# B&R Automation Studio project RS15_RX_30005_r00 (part 10)

#### HGWeber.fun - Exported functions and function blocks
```iecst
(********************************************************************
 * COPYRIGHT --
 ********************************************************************
 * Library: HGWeber
 * File: HGWeber.fun
 * Author: pkiel
 * Created: September 03, 2009
 ********************************************************************
 * Functions and function blocks of library HGWeber
 ********************************************************************)

FUNCTION H_FC_Modulus_V0 : REAL  (*Calculat the modulus of number*)
  VAR_INPUT
    IN_rMod : REAL ;
    IN_rVar : REAL ;
  END_VAR
  VAR
    rVar : REAL;
  END_VAR
END_FUNCTION

FUNCTION H_FC_Modulus : REAL  (*Calculat the modulus of number*)
  VAR_INPUT
    IN_rMod : REAL ;
    IN_rVar : REAL ;
  END_VAR
  VAR
    rVar : REAL;
  END_VAR
END_FUNCTION

FUNCTION_BLOCK HGW_2StatePB (*Two State Pushbutton Control/Indication*)
	VAR_INPUT
		PB : BOOL; (*Add your parameter comment*)
		Reset : BOOL; (*Add your parameter comment*)
		BackColor_State0 : UINT; (*Add your parameter comment*)
		ForeColor_State0 : UINT; (*Add your parameter comment*)
		BackColor_State1 : UINT; (*Add your parameter comment*)
		ForeColor_State1 : UINT; (*Add your parameter comment*)
	END_VAR
	VAR_OUTPUT
		Text_Ind : UINT; (*Add your parameter comment*)
		Color_Ind : UINT; (*Add your parameter comment*)
		State0 : BOOL; (*Add your parameter comment*)
		State1 : BOOL; (*Add your parameter comment*)
	END_VAR
	VAR
		R_Trig1 : r_trig;
	END_VAR
END_FUNCTION_BLOCK

FUNCTION_BLOCK HGW_3StatePB (*Three State Pushbutton Control/Indication*)
	VAR_INPUT
		PB : BOOL; (*Add your parameter comment*)
		Reset : BOOL; (*Add your parameter comment*)
		BackColor_State0 : UINT; (*Add your parameter comment*)
		ForeColor_State0 : UINT; (*Add your parameter comment*)
		BackColor_State1 : UINT; (*Add your parameter comment*)
		ForeColor_State1 : UINT; (*Add your parameter comment*)
		BackColor_State2 : UINT;
		ForeColor_State2 : UINT;
	END_VAR
	VAR_OUTPUT
		Text_Ind : UINT; (*Add your parameter comment*)
		Color_Ind : UINT; (*Add your parameter comment*)
		State0 : BOOL; (*Add your parameter comment*)
		State1 : BOOL; (*Add your parameter comment*)
		State2 : BOOL; (*Add your parameter comment*)
	END_VAR
	VAR
		R_Trig1 : r_trig;
	END_VAR
END_FUNCTION_BLOCK

FUNCTION_BLOCK HGW_4StatePB (*Four State Pushbutton Control/Indication*)
	VAR_INPUT
		PB : BOOL; (*Add your parameter comment*)
		Reset : BOOL; (*Add your parameter comment*)
		BackColor_State0 : UINT; (*Add your parameter comment*)
		ForeColor_State0 : UINT; (*Add your parameter comment*)
		BackColor_State1 : UINT; (*Add your parameter comment*)
		ForeColor_State1 : UINT; (*Add your parameter comment*)
		BackColor_State2 : UINT; (*Add your parameter comment*)
		ForeColor_State2 : UINT; (*Add your parameter comment*)
		BackColor_State3 : UINT; (*Add your parameter comment*)
		ForeColor_State3 : UINT; (*Add your parameter comment*)
	END_VAR
	VAR_OUTPUT
		Text_Ind : UINT; (*Add your parameter comment*)
		Color_Ind : UINT; (*Add your parameter comment*)
		State0 : BOOL; (*Add your parameter comment*)
		State1 : BOOL; (*Add your parameter comment*)
		State2 : BOOL; (*Add your parameter comment*)
		State3 : BOOL; (*Add your parameter comment*)
	END_VAR
	VAR
		R_Trig1 : r_trig;
	END_VAR
END_FUNCTION_BLOCK

FUNCTION_BLOCK HGW_2StateIND (*Two State Indication*)
	VAR_INPUT
		In_State : BOOL; (*Add your parameter comment*)
		BackColor_State0 : UINT; (*Add your parameter comment*)
		ForeColor_State0 : UINT; (*Add your parameter comment*)
		BackColor_State1 : UINT; (*Add your parameter comment*)
		ForeColor_State1 : UINT; (*Add your parameter comment*)
	END_VAR
	VAR_OUTPUT
		Text_Ind : UINT; (*Add your parameter comment*)
		Color_Ind : UINT; (*Add your parameter comment*)
		State0 : BOOL; (*Add your parameter comment*)
		State1 : BOOL; (*Add your parameter comment*)
	END_VAR
END_FUNCTION_BLOCK

FUNCTION_BLOCK HGW_3StateIND (*Three State Indication*)
  VAR_INPUT
    In_State0 : BOOL; (*Add your parameter comment*)
    In_State1 : BOOL; (*Add your parameter comment*)
    In_State2 : BOOL; (*Add your parameter comment*)
    BackColor_State0 : UINT; (*Add your parameter comment*)
    ForeColor_State0 : UINT; (*Add your parameter comment*)
    BackColor_State1 : UINT; (*Add your parameter comment*)
    ForeColor_State1 : UINT; (*Add your parameter comment*)
    BackColor_State2 : UINT; (*Add your parameter comment*)
    ForeColor_State2 : UINT; (*Add your parameter comment*)
  END_VAR
  VAR_OUTPUT
    Text_Ind : UINT; (*Add your parameter comment*)
    Color_Ind : UINT; (*Add your parameter comment*)
    State0 : BOOL; (*Add your parameter comment*)
    State1 : BOOL; (*Add your parameter comment*)
    State2 : BOOL; (*Add your parameter comment*)
  END_VAR
END_FUNCTION_BLOCK

FUNCTION_BLOCK HGW_3StateIND1 (*Three State Indication*)
  VAR_INPUT
    IN_bState0 : BOOL; (*Add your parameter comment*)
    IN_bState1 : BOOL; (*Add your parameter comment*)
    IN_bState2 : BOOL; (*Add your parameter comment*)
    IN_bFlash  : BOOL; (*Add your parameter comment*)
    IN_uiTxt_Ind_State0 : UINT := 0 ;
    IN_uiTxt_Ind_State1 : UINT := 1 ;
    IN_uiTxt_Ind_State2 : UINT := 2 ;
    IN_rNumFlashPerSec  : REAL := 1 ; (*Number of flash per second*)
    IN_uiBackCol_State0 : UINT; (*Add your parameter comment*)
    IN_uiForeCol_State0 : UINT; (*Add your parameter comment*)
    IN_uiBackCol_State1 : UINT; (*Add your parameter comment*)
    IN_uiForeCol_State1 : UINT; (*Add your parameter comment*)
    IN_uiBackCol_State2 : UINT; (*Add your parameter comment*)
    IN_uiForeCol_State2 : UINT; (*Add your parameter comment*)
    IN_uiBackColFlash_Off_State0 : UINT; (*Add your parameter comment*)
    IN_uiForeColFlash_Off_State0 : UINT; (*Add your parameter comment*)
    IN_uiBackColFlash_On_State0  : UINT; (*Add your parameter comment*)
    IN_uiForeColFlash_On_State0  : UINT; (*Add your parameter comment*)
    IN_uiBackColFlash_Off_State1 : UINT; (*Add your parameter comment*)
    IN_uiForeColFlash_Off_State1 : UINT; (*Add your parameter comment*)
    IN_uiBackColFlash_On_State1  : UINT; (*Add your parameter comment*)
    IN_uiForeColFlash_On_State1  : UINT; (*Add your parameter comment*)
    IN_uiBackColFlash_Off_State2 : UINT; (*Add your parameter comment*)
    IN_uiForeColFlash_Off_State2 : UINT; (*Add your parameter comment*)
    IN_uiBackColFlash_On_State2  : UINT; (*Add your parameter comment*)
    IN_uiForeColFlash_On_State2  : UINT; (*Add your parameter comment*)

  END_VAR
  VAR_OUTPUT
    OUT_uiTxt_Ind : UINT; (*Add your parameter comment*)
    OUT_uiCol_Ind : UINT; (*Add your parameter comment*)
    OUT_bState0   : BOOL; (*Add your parameter comment*)
    OUT_bState1   : BOOL; (*Add your parameter comment*)
    OUT_bState2   : BOOL; (*Add your parameter comment*)
  END_VAR
  VAR
    stTON_1  : TON;
    stTON_0  : TON;
    bFlash   : BOOL;
    tTpFlash : TIME ;
  END_VAR
END_FUNCTION_BLOCK
FUNCTION_BLOCK HGW_4StateIND (*Four State Indication*)
	VAR_INPUT
		In_State0 : BOOL; (*Add your parameter comment*)
		In_State1 : BOOL; (*Add your parameter comment*)
		In_State2 : BOOL; (*Add your parameter comment*)
		In_State3 : BOOL; (*Add your parameter comment*)
		BackColor_State0 : UINT; (*Add your parameter comment*)
		ForeColor_State0 : UINT; (*Add your parameter comment*)
		BackColor_State1 : UINT; (*Add your parameter comment*)
		ForeColor_State1 : UINT; (*Add your parameter comment*)
		BackColor_State2 : UINT; (*Add your parameter comment*)
		ForeColor_State2 : UINT; (*Add your parameter comment*)
		BackColor_State3 : UINT; (*Add your parameter comment*)
		ForeColor_State3 : UINT; (*Add your parameter comment*)
	END_VAR
	VAR_OUTPUT
		Text_Ind : UINT; (*Add your parameter comment*)
		Color_Ind : UINT; (*Add your parameter comment*)
		State0 : BOOL; (*Add your parameter comment*)
		State1 : BOOL; (*Add your parameter comment*)
		State2 : BOOL; (*Add your parameter comment*)
		State3 : BOOL; (*Add your parameter comment*)
	END_VAR
END_FUNCTION_BLOCK

FUNCTION_BLOCK HGW_Toggle (*Time Based Toggle For Bool*)
	VAR_INPUT
		In : BOOL; (*Add your parameter comment*)
		Time : TIME; (*Add your parameter comment*)
	END_VAR
	VAR_OUTPUT
		Out : BOOL; (*Add your parameter comment*)
	END_VAR
	VAR
		zzInternalMemory : ARRAY[0..9] OF SINT; (*Internal memory*)
		TON_0 : TON; (*Add your parameter comment*)
		TON_1 : TON; (*Add your parameter comment*)
	END_VAR
END_FUNCTION_BLOCK

FUNCTION_BLOCK HGW_2StepMove (*Standard Two Step Move*)
  VAR_INPUT
    MoveRequest : BOOL; (*Add your parameter comment*)
    Permissive  : BOOL; (*Add your parameter comment*)
  END_VAR
  VAR_OUTPUT
    Horn : BOOL; (*Add your parameter comment*)
    StartMove : BOOL; (*Add your parameter comment*)
  END_VAR
  VAR
    HornDone : BOOL; (*Add your parameter comment*)
    StartWindow : BOOL; (*Add your parameter comment*)
    TON_0 : TON; (*Add your parameter comment*)
    TON_1 : TON; (*Add your parameter comment*)
    TON_2 : TON; (*Add your parameter comment*)
    zzInternalMemory : ARRAY[0..9] OF SINT; (*Internal memory*)
  END_VAR
END_FUNCTION_BLOCK

FUNCTION_BLOCK HGW_ChangeReal (*Detects A Change Of A Real Number For One Scan*)
	VAR_INPUT
		Enable : BOOL; (*Add your parameter comment*)
		Input : REAL; (*Add your parameter comment*)
	END_VAR
	VAR_OUTPUT
		OK : BOOL; (*Add your parameter comment*)
		Change : BOOL; (*Add your parameter comment*)
	END_VAR
	VAR
		Old : REAL; (*Add your parameter comment*)
	END_VAR
END_FUNCTION_BLOCK

FUNCTION_BLOCK HGW_ScaleReal (*Scales A Real Value A Scaled Range*)
	VAR_INPUT
		Enable : BOOL; (*Add your parameter comment*)
		InputMin : REAL; (*Add your parameter comment*)
		InputMax : REAL; (*Add your parameter comment*)
		InputRaw : REAL; (*Add your parameter comment*)
		ScaledMin : REAL; (*Add your parameter comment*)
		ScaledMax : REAL; (*Add your parameter comment*)
	END_VAR
	VAR_OUTPUT
		OK : BOOL; (*Add your parameter comment*)
		ScaledOut : REAL; (*Add your parameter comment*)
		Error : BOOL; (*Add your parameter comment*)
	END_VAR
	VAR
		InputDiff : REAL; (*Add your parameter comment*)
		ScaledDiff : REAL; (*Add your parameter comment*)
		Slope : REAL; (*Add your parameter comment*)
		Offset : REAL; (*Add your parameter comment*)
	END_VAR
END_FUNCTION_BLOCK

FUNCTION_BLOCK HGW_RelativeChangeReal (*Detects A Change Of A Real Variable & Outputs the Relative Change*)
	VAR_INPUT
		Enable : BOOL; (*Add your parameter comment*)
		Input : REAL; (*Add your parameter comment*)
	END_VAR
	VAR_OUTPUT
		OK : BOOL; (*Add your parameter comment*)
		Change : BOOL; (*Add your parameter comment*)
		Diff : REAL; (*Add your parameter comment*)
	END_VAR
	VAR
		Old : REAL; (*Add your parameter comment*)
	END_VAR
END_FUNCTION_BLOCK

FUNCTION_BLOCK HGW_Average (*Running/Weighted Averaging Of A Real Value*)
	VAR_INPUT
		Enable : BOOL; (*Add your parameter comment*)
		Execute : BOOL; (*Add your parameter comment*)
		ProgramLength : REAL; (*Add your parameter comment*)
		ActualLength : REAL; (*Add your parameter comment*)
	END_VAR
	VAR_OUTPUT
		AverageLength : REAL; (*Add your parameter comment*)
		Update : BOOL; (*Add your parameter comment*)
	END_VAR
	VAR
		R_Trig0 : r_trig; (*Add your parameter comment*)
		R_Trig1 : r_trig; (*Add your parameter comment*)
		Count : INT; (*Add your parameter comment*)
		Accum : REAL; (*Add your parameter comment*)
		Length : REAL; (*Add your parameter comment*)
	END_VAR
END_FUNCTION_BLOCK

FUNCTION_BLOCK HGW_RegCorrectABS (*Calculates Registration Correction For Absolute Type Registration*)
	VAR_INPUT
		Enable : BOOL; (*Add your parameter comment*)
		Execute : BOOL; (*Add your parameter comment*)
		NewCapture : REAL; (*Add your parameter comment*)
		Expected : REAL; (*Add your parameter comment*)
		Period : REAL; (*Add your parameter comment*)
		WeightingFactor : REAL; (*Add your parameter comment*)
		MaxCorrection : REAL; (*Add your parameter comment*)
	END_VAR
	VAR_OUTPUT
		OK : BOOL; (*Add your parameter comment*)
		Correction : REAL; (*Add your parameter comment*)
		MaxCorrectionExceeded : BOOL; (*Add your parameter comment*)
	END_VAR
	VAR
		R_Trig0 : r_trig; (*Add your parameter comment*)
		R_Trig1 : r_trig; (*Add your parameter comment*)
		Max_Positive : BOOL;
		Max_Negative : BOOL;
	END_VAR
END_FUNCTION_BLOCK

FUNCTION_BLOCK HGW_KeyRepeat (*Toggles A Bool At A Rate After An Initial Delay*)
	VAR_INPUT
		Key_In : BOOL; (*Add your parameter comment*)
		Delay : TIME; (*Add your parameter comment*)
		Rate : TIME; (*Add your parameter comment*)
	END_VAR
	VAR_OUTPUT
		Key_Out : BOOL; (*Add your parameter comment*)
	END_VAR
	VAR
		TON_0 : TON; (*Add your parameter comment*)
		TON_1 : TON; (*Add your parameter comment*)
		TON_2 : TON; (*Add your parameter comment*)
		R_Trig0 : r_trig; (*Add your parameter comment*)
		R_Trig1 : r_trig; (*Add your parameter comment*)
		R_Trig2 : r_trig;
	END_VAR
END_FUNCTION_BLOCK

FUNCTION_BLOCK HGW_2StateIND1 (*Two State Indication With "0" State Flash*)
	VAR_INPUT
		In_State : BOOL; (*Add your parameter comment*)
		BackColorFlash_Off : UINT; (*Add your parameter comment*)
		ForeColorFlash_Off : UINT; (*Add your parameter comment*)
		BackColorFlash_On : UINT; (*Add your parameter comment*)
		ForeColorFlash_On : UINT; (*Add your parameter comment*)
		BackColor_State1 : UINT; (*Add your parameter comment*)
		ForeColor_State1 : UINT; (*Add your parameter comment*)
	END_VAR
	VAR_OUTPUT
		Text_Ind : UINT; (*Add your parameter comment*)
		Color_Ind : UINT; (*Add your parameter comment*)
		State0 : BOOL; (*Add your parameter comment*)
		State1 : BOOL; (*Add your parameter comment*)
	END_VAR
	VAR
		TON_1 : TON;
		TON_0 : TON;
		Flash : BOOL;
	END_VAR

END_FUNCTION_BLOCK

FUNCTION_BLOCK HGW_2StepMove1  (*TODO: Add your comment here*)

  VAR_INPUT
    IN_bMoveRequest : BOOL; (*Add your parameter comment*)
    IN_bPermissive  : BOOL; (*Add your parameter comment*)
    IN_bCasRun      : BOOL := 0; (*=1 case Run, =0 case Jog*)
    IN_tTpHorn      : TIME; (*Horn duration, in s*)
  END_VAR
  VAR_OUTPUT
    OUT_bHorn : BOOL; (*Add your parameter comment*)
    OUT_bStartMove : BOOL; (*Add your parameter comment*)
  END_VAR
  VAR
    tTimReset : TIME; (*Add your parameter comment*)
    bHornDone : BOOL; (*Add your parameter comment*)
    bStartWindow : BOOL; (*Add your parameter comment*)
    stTON_0 : TON; (*Add your parameter comment*)
    stTON_1 : TON; (*Add your parameter comment*)
    stTON_2 : TON; (*Add your parameter comment*)
    zzInternalMemory : ARRAY[0..12] OF SINT; (*Internal memory*)
  END_VAR
END_FUNCTION_BLOCK

FUNCTION_BLOCK H_FB_2StepMove  (*TODO: Add your comment here*)

  VAR_INPUT
    IN_bStart  : BOOL ;  (**)
    IN_bPermis : BOOL ;
    IN_tTpHorn : TIME ;
  END_VAR
  VAR_OUTPUT
    OUT_bHorn      : BOOL ;  (**)
    OUT_bStartMove : BOOL ;  (**)
    OUT_iActStep   : INT ;
  END_VAR
  VAR_IN_OUT
  END_VAR
  VAR
    stTON_0 : TON ;  (**)
    stTON_1 : TON ;  (**)
    stTON_2 : TON ;  (**)
    stTON_3 : TON ;  (**)
    iStep   : INT ;
    zzEdge00000 : BOOL;
    zzEdge00001 : BOOL;
  END_VAR
END_FUNCTION_BLOCK

FUNCTION_BLOCK H_FB_ToggleTB  (*TODO: Add your comment here*)

  VAR_INPUT
    IN_bTB : BOOL ;  (**)
    IN_uiTxt1_Ind       : INT ;
    IN_uiTxt0_Ind       : INT ;
    IN_uiBackCol_State0 : UINT; (*Add your parameter comment*)
    IN_uiForeCol_State0 : UINT; (*Add your parameter comment*)
    IN_uiBackCol_State1 : UINT; (*Add your parameter comment*)
    IN_uiForeCol_State1 : UINT; (*Add your parameter comment*)
  END_VAR
  VAR_OUTPUT
    OUT_uiTxt_Ind : UINT; (*Add your parameter comment*)
    OUT_uiCol_Ind : UINT; (*Add your parameter comment*)
  END_VAR
  VAR_IN_OUT
  END_VAR
  VAR
    zzEdge00000 : BOOL;
  END_VAR
END_FUNCTION_BLOCK

FUNCTION_BLOCK H_FB_WatchSensor  (*TODO: Add your comment here*)

  VAR_INPUT
    IN_bActSensIn       : BOOL ; (*Act watch sensor In*)
    IN_bSensorIn        : BOOL := 0 ;
    IN_bActSensOut      : BOOL ; (*Act watch sensor Out*)
    IN_bSensorOut       : BOOL := 0 ;
    IN_bSOL_In          : BOOL := 0 ;
    IN_bSOL_Out         : BOOL := 0 ;
    IN_bReset           : BOOL ;
    IN_tTpWatchIn       : TIME := T#4s ; (*Default time =4s*)
    IN_tTpWatchOut      : TIME := T#4s ; (*Default time =4s*)
    IN_tTpFiltDI        : TIME := T#30ms ; (*Time filtering input sensor default time =30ms*)
  END_VAR
  VAR_OUTPUT
    OUT_bSensIn_FaultIn   : BOOL ; (*Add your parameter comment*)
    OUT_bSensIn_FaultOut  : BOOL ; (*Add your parameter comment*)
    OUT_bSensOut_FaultIn  : BOOL ; (*Add your parameter comment*)
    OUT_bSensOut_FaultOut : BOOL ; (*Add your parameter comment*)
    OUT_bSensIn_Fault     : BOOL ; (*Add your parameter comment*)
    OUT_bSensOut_Fault    : BOOL ; (*Add your parameter comment*)
    OUT_bSens_Fault       : BOOL ; (*Add your parameter comment*)
  END_VAR
  VAR_IN_OUT
  END_VAR
  VAR
    bReset  : BOOL ;
    bSensorIn     : BOOL ;
    bSensorOut    : BOOL ;
    stTON_SOL_Out : TON ;
    stTON_SOL_In  : TON ;
    stTON_FiltSensIn  : TON ;
    stTOF_FiltSensIn  : TOF ;
    stTON_FiltSensOut : TON ;
    stTOF_FiltSensOut : TOF ;
    zzEdge00000 : BOOL;
  END_VAR
END_FUNCTION_BLOCK

FUNCTION_BLOCK H_FB_Flash  (*TODO: Add your comment here*)

  VAR_INPUT
    IN_bEnable          : BOOL ;
    IN_rNumFlashPerSec  : REAL := 1 ; (*Number of flash per second*)
  END_VAR
  VAR_OUTPUT
    OUT_bFlash : BOOL ; (*Add your parameter comment*)
  END_VAR
  VAR
    tTpFlash : TIME ;
    stTON_0  : TON ;
    stTON_1  : TON ;
    zzEdge00000 : BOOL;
  END_VAR
END_FUNCTION_BLOCK

FUNCTION_BLOCK H_FB_RelativeChangeLimitReal  (*TODO: Add your comment here*)
  VAR_INPUT
    IN_bEnable : BOOL; (*Add your parameter comment*)
    IN_rMax    : REAL;
    IN_rMin    : REAL;
    IN_rInput  : REAL;
    IN_rRepeat : REAL;
  END_VAR
  VAR_IN_OUT
    INOUT_rLimitIn : REAL; (*Limited input*)
  END_VAR
  VAR_OUTPUT
    OUT_bOK : BOOL; (*Add your parameter comment*)
    OUT_bChange : BOOL; (*Add your parameter comment*)
    OUT_rDiff : REAL; (*Add your parameter comment*)
  END_VAR
  VAR
    rInput : REAL; (*Add your parameter comment*)
    rOld   : REAL; (*Add your parameter comment*)
    rDiff  : REAL; (*Add your parameter comment*)
    rMax   : REAL; (*Add your parameter comment*)
    rMin   : REAL; (*Add your parameter comment*)
    rOldLimitIn : REAL; (*Add your parameter comment*)
    rLimitIn    : REAL; (*Add your parameter comment*)
  END_VAR
END_FUNCTION_BLOCK

FUNCTION_BLOCK H_FB_RelativeChangeLimitReal1  (*TODO: Add your comment here*)
  VAR_INPUT
    IN_bEnable : BOOL; (*Add your parameter comment*)
    IN_rMax    : REAL;
    IN_rMin    : REAL;
    IN_rInput  : REAL;
    IN_rRepeat : REAL;
    IN_rLimitIn : REAL; (*Limited input*)
  END_VAR
  VAR_IN_OUT
  END_VAR
  VAR_OUTPUT
    OUT_bOK : BOOL; (*Add your parameter comment*)
    OUT_bChange : BOOL; (*Add your parameter comment*)
    OUT_rDiff : REAL; (*Add your parameter comment*)
    OUT_rLimitIn : REAL; (*Limited input*)
  END_VAR
  VAR
    rInput : REAL; (*Add your parameter comment*)
    rOld   : REAL; (*Add your parameter comment*)
    rDiff  : REAL; (*Add your parameter comment*)
    rMax   : REAL; (*Add your parameter comment*)
    rMin   : REAL; (*Add your parameter comment*)
    rOldLimitIn : REAL; (*Add your parameter comment*)
    iCount : INT ;
  END_VAR
END_FUNCTION_BLOCK
```

#### HGW_2StatePB.st - Two State Pushbutton Control/Indication
```iecst
(********************************************************************
 * COPYRIGHT --
 ********************************************************************
 * Library: HGWeber
 * File: HGW_2StatePB.st
 * Author: pkiel
 * Created: September 03, 2009
 ********************************************************************
 * Implementation of library HGWeber
 ********************************************************************)

(*Two State Pushbutton Control/Indication*)
FUNCTION_BLOCK HGW_2StatePB

	R_Trig1(CLK:=PB);
	IF(R_Trig1.Q)THEN
		Text_Ind := 1 + Text_Ind;
	END_IF
	IF (Reset) THEN
		Text_Ind :=0;
	END_IF

	(* For Each Button Press, the internal state is changed...changing the text, color, and state indications *)

	CASE Text_Ind OF
		0:
			Color_Ind := BackColor_State0 + ForeColor_State0 * 256;
			State0 := 1;
			State1 := 0;
		1:
			Color_Ind := BackColor_State1 + ForeColor_State1 * 256;
			State0 := 0;
			State1 := 1;
		2:
			Text_Ind := 0;
	END_CASE

END_FUNCTION_BLOCK
```

#### HGW_2StateIND1.st - Two State Indication With "0" State Flash
```iecst
(********************************************************************
 * COPYRIGHT --
 ********************************************************************
 * Library: HGWeber
 * File: HGW_2StateIND1.st
 * Author: pkiel
 * Created: October 13, 2009
 ********************************************************************
 * Implementation of library HGWeber
 ********************************************************************)

(*Two State Indication With "0" State Flash*)
FUNCTION_BLOCK HGW_2StateIND1

	IF(In_State)THEN
		Text_Ind := 1;
	ELSE
		Text_Ind := 0;
	END_IF

	TON_0(IN:=NOT(TON_1.Q),PT:=T#1s );
	TON_1(IN:=TON_0.Q,PT:=T#1s);
	Flash:=TON_0.Q;

	CASE Text_Ind OF
		0:
			IF (Flash) THEN
				Color_Ind := BackColorFlash_On + ForeColorFlash_On * 256;
			ELSE
				Color_Ind := BackColorFlash_Off + ForeColorFlash_Off * 256;
			END_IF
			State0 := 1;
			State1 := 0;
		1:
			Color_Ind := BackColor_State1 + ForeColor_State1 * 256;
			State0 := 0;
			State1 := 1;
		2:
			Text_Ind := 0;
	END_CASE

END_FUNCTION_BLOCK
```

#### HGW_3StateIND1.st - Three State Indication
```iecst
(********************************************************************
 * COPYRIGHT --
 ********************************************************************
 * Library: HGWeber
 * File: HGW_3StateIND.st
 * Author: pkiel
 * Created: September 03, 2009
 ********************************************************************
 * Implementation of library HGWeber
 ********************************************************************)

(*Three State Indication*)
FUNCTION_BLOCK HGW_3StateIND1

	IF(IN_bState0)THEN
		OUT_uiTxt_Ind := IN_uiTxt_Ind_State0 ;
	END_IF
	IF(IN_bState1)THEN
		OUT_uiTxt_Ind := IN_uiTxt_Ind_State1 ;
	END_IF
	IF(IN_bState2)THEN
		OUT_uiTxt_Ind := IN_uiTxt_Ind_State2 ;
	END_IF

  tTpFlash := REAL_TO_TIME(1000/IN_rNumFlashPerSec) ;
  stTON_0(IN:=NOT(stTON_1.Q),PT:=tTpFlash);
  stTON_1(IN:=stTON_0.Q,PT:=tTpFlash);
  bFlash:=stTON_0.Q;

	CASE OUT_uiTxt_Ind OF
		0:
      IF IN_bFlash THEN
        IF (bFlash) THEN
          OUT_uiCol_Ind := IN_uiBackColFlash_On_State0 + IN_uiForeColFlash_On_State0 * 256;
        ELSE
          OUT_uiCol_Ind := IN_uiBackColFlash_Off_State0 + IN_uiForeColFlash_Off_State0 * 256;
        END_IF
      ELSE
        OUT_uiCol_Ind := IN_uiBackCol_State0 + IN_uiForeCol_State0 * 256;
      END_IF
			OUT_bState0 := 1;
			OUT_bState1 := 0;
			OUT_bState2 := 0;
		1:
      IF IN_bFlash THEN
        IF (bFlash) THEN
          OUT_uiCol_Ind := IN_uiBackColFlash_On_State1 + IN_uiForeColFlash_On_State1 * 256;
        ELSE
          OUT_uiCol_Ind := IN_uiBackColFlash_Off_State1 + IN_uiForeColFlash_Off_State1 * 256;
        END_IF
      ELSE
        OUT_uiCol_Ind := IN_uiBackCol_State1 + IN_uiForeCol_State1 * 256;
      END_IF
			OUT_bState0 := 0;
			OUT_bState1 := 1;
			OUT_bState2 := 0;
		2:
      IF IN_bFlash THEN
        IF (bFlash) THEN
          OUT_uiCol_Ind := IN_uiBackColFlash_On_State2 + IN_uiForeColFlash_On_State2 * 256;
        ELSE
          OUT_uiCol_Ind := IN_uiBackColFlash_Off_State2 + IN_uiForeColFlash_Off_State2 * 256;
        END_IF
      ELSE
        OUT_uiCol_Ind := IN_uiBackCol_State2 + IN_uiForeCol_State2 * 256;
      END_IF
			OUT_bState0 := 0;
			OUT_bState1 := 0;
			OUT_bState2 := 1;
		3:
			OUT_uiTxt_Ind := 0;
	END_CASE

END_FUNCTION_BLOCK
```

#### HGW_ChangeReal.st - Detects A Change Of A Real Number For One Scan
```iecst
(********************************************************************
 * COPYRIGHT --
 ********************************************************************
 * Library: HGWeber
 * File: HGW_ChangeReal.st
 * Author: pkiel
 * Created: September 03, 2009
 ********************************************************************
 * Implementation of library HGWeber
 ********************************************************************)

(*Detects A Change Of A Real Number For One Scan*)
FUNCTION_BLOCK HGW_ChangeReal

	OK := Enable;
	IF (Enable) THEN
		IF (Input <> Old) THEN
			Change := 1;
			Old := Input;
		ELSE
			Change := 0;
		END_IF
	ELSE;
		Change :=0;
	END_IF;

END_FUNCTION_BLOCK
```

#### HGW_RelativeChangeReal.st - Detects A Change Of A Real Variable & Outputs the Relative Change
```iecst
(********************************************************************
 * COPYRIGHT --
 ********************************************************************
 * Library: HGWeber
 * File: HGW_RelativeChangeReal.st
 * Author: pkiel
 * Created: September 03, 2009
 ********************************************************************
 * Implementation of library HGWeber
 ********************************************************************)

(*Detects A Change Of A Real Variable & Outputs the Relative Change*)
FUNCTION_BLOCK HGW_RelativeChangeReal

	OK := Enable;
	IF (Enable) THEN
		IF (Input <> Old) THEN
			Change := 1;
			Diff := Input-Old;
			Old := Input;
		ELSE
			Change := 0;
		END_IF
	ELSE
		Change :=0;
	END_IF

END_FUNCTION_BLOCK
```

#### HGW_Average.st - Running/Weighted Averaging Of A Real Value
```iecst
(********************************************************************
 * COPYRIGHT --
 ********************************************************************
 * Library: HGWeber
 * File: HGW_Average.st
 * Author: pkiel
 * Created: September 03, 2009
 ********************************************************************
 * Implementation of library HGWeber
 ********************************************************************)

(*Running/Weighted Averaging Of A Real Value*)
FUNCTION_BLOCK HGW_Average

	R_Trig0 (CLK:=Enable);
	IF (R_Trig0.Q) THEN
		AverageLength:=ProgramLength;
		Count:=0;
		Accum:=0;
	END_IF;

	R_Trig1 (CLK:=Execute);
	IF (R_Trig1.Q) THEN
		Length:=LIMIT(0.99*ProgramLength,ActualLength,1.01*ProgramLength);
		Accum:=Accum+Length;
		Count:=Count+1;
		AverageLength:=Accum/Count;
	END_IF;
	IF (Count>=24) THEN
		Count:=Count/2;
		Accum:=Accum/2;
		Update:=1;
	ELSE;
		Update:=0;
	END_IF;

END_FUNCTION_BLOCK
```

#### HGW_RegCorrectABS.st - Calculates Registration Correction For Absolute Type Registration
```iecst
(********************************************************************
 * COPYRIGHT --
 ********************************************************************
 * Library: HGWeber
 * File: HGW_RegCorrectABS.st
 * Author: pkiel
 * Created: September 03, 2009
 ********************************************************************
 * Implementation of library HGWeber
 ********************************************************************)

(*Calculates Registration Correction For Absolute Type Registration*)
FUNCTION_BLOCK HGW_RegCorrectABS

	OK := Enable;

	(*Zero Out Correction Value When First Enabled*)
	R_Trig0 (CLK:= Enable);
	IF (R_Trig0.Q) THEN
		Correction :=0;
	END_IF

	(*Calculate Correction*)
	R_Trig1 (CLK:= Execute);
	IF (R_Trig1.Q) THEN
		Correction := Expected-NewCapture;
		IF (Correction>(Period/2.0)) THEN
			Correction := Correction-Period;
		END_IF
		IF (Correction<(-Period/2.0)) THEN
			Correction := Correction+Period;
		END_IF
	Correction := -WeightingFactor*Correction;
	END_IF

	(*Evaluate Correction For Limits*)
	IF (Correction>MaxCorrection) THEN
		Correction := MaxCorrection;
		Max_Positive := 1;
	ELSE;
		Max_Positive := 0;
	END_IF

	IF (Correction<-MaxCorrection) THEN
		Correction := -MaxCorrection;
		Max_Negative := 1;
	ELSE;
		Max_Negative := 0;
	END_IF;

	IF (Max_Positive OR Max_Negative) THEN
		MaxCorrectionExceeded := 1;
	ELSE;
		MaxCorrectionExceeded := 0;
	END_IF;

END_FUNCTION_BLOCK
```

#### HGW_2StepMove1.ld
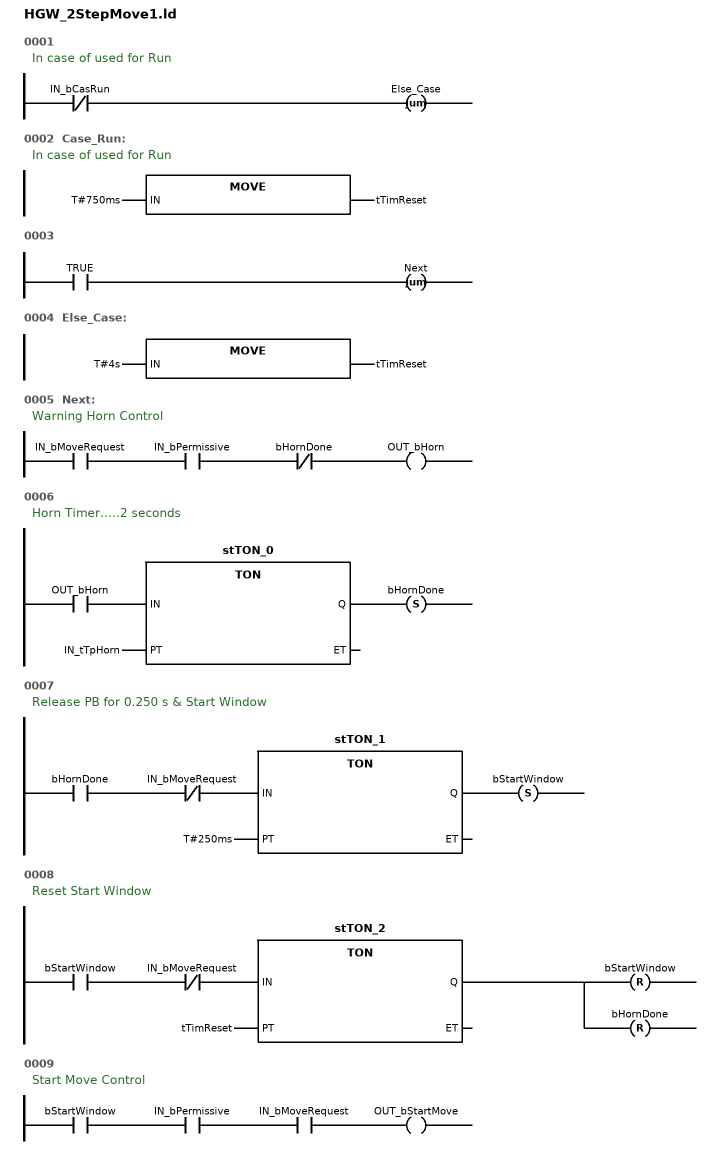
Ladder, written as Structured Text:
```iecst
FUNCTION_BLOCK HGW_2StepMove1
(* Network 1: In case of used for Run  *)
IF NOT IN_bCasRun THEN JMP Else_Case; END_IF;

(* Network 2: In case of used for Run  *)
Case_Run:
tTimReset := T#750ms;

(* Network 3 *)
JMP Next;

(* Network 4 *)
Else_Case:
tTimReset := T#4s;

(* Network 5: Warning Horn Control *)
Next:
OUT_bHorn := IN_bMoveRequest AND IN_bPermissive AND NOT bHornDone;

(* Network 6: Horn Timer.....2 seconds *)
stTON_0(IN := OUT_bHorn, PT := IN_tTpHorn);
IF stTON_0.Q THEN bHornDone := TRUE; END_IF;

(* Network 7: Release PB for 0.250 s & Start Window *)
stTON_1(IN := bHornDone AND NOT IN_bMoveRequest, PT := T#250ms);
IF stTON_1.Q THEN bStartWindow := TRUE; END_IF;

(* Network 8: Reset Start Window *)
stTON_2(IN := bStartWindow AND NOT IN_bMoveRequest, PT := tTimReset);
IF stTON_2.Q THEN
    bStartWindow := FALSE;
    bHornDone := FALSE;
END_IF;

(* Network 9: Start Move Control *)
OUT_bStartMove := bStartWindow AND IN_bPermissive AND IN_bMoveRequest;
END_FUNCTION_BLOCK
```

#### H_FB_Flash.st
```iecst
(********************************************************************
 * COPYRIGHT -- .
 ********************************************************************
 * Library: HGWeber
 * File: H_FB_Flash.st
 * Author: dominique
 * Created: August 19, 2011
 ********************************************************************
 * Implementation of library HGWeber
 ********************************************************************)

FUNCTION_BLOCK H_FB_Flash

  IF IN_bEnable THEN
    tTpFlash := REAL_TO_TIME(1000/IN_rNumFlashPerSec) ;
    stTON_0(IN:=NOT(stTON_1.Q),PT:=tTpFlash);
    stTON_1(IN:=stTON_0.Q,PT:=tTpFlash);

    OUT_bFlash:=stTON_0.Q ;
  ELSE
    OUT_bFlash:= 0 ;
  END_IF ;

END_FUNCTION_BLOCK
```

#### H_FB_RelativeChangeLimitReal.st - Detects A Change Of A Real Number For One Scan
```iecst
(********************************************************************
 * COPYRIGHT --
 ********************************************************************
 * Library: HGWeber
 * File: H_FB_RelativeChangeLimitReal.st
 * Author: dominique
 * Created: October 10, 2011
 ********************************************************************
 * Implementation of library HGWeber
 ********************************************************************)

(*Detects A Change Of A Real Number For One Scan and limit the Change*)
FUNCTION_BLOCK H_FB_RelativeChangeLimitReal

  // D.M. 11/10/2011 BrownPaper_14543  FB not usable. VAR_IN_OUT does no work at all... contains always a big value no idea where it come from and not possible to write it...

  rMax     := IN_rRepeat * IN_rMax ;
  rMin     := IN_rRepeat * IN_rMin ;
  rLimitIn := INOUT_rLimitIn ;

	OUT_bOK := IN_bEnable;
	IF (IN_bEnable) THEN
    rDiff := rLimitIn - rOldLimitIn ;
    // Limit relative change
    IF rDiff > rMax THEN
      rLimitIn := rOldLimitIn + rMax ;
    END_IF
    IF rDiff < rMin THEN
      rLimitIn := rOldLimitIn + rMin ;
    END_IF
    rInput := rLimitIn + IN_rInput ;
		IF (rInput <> rOld) THEN
			OUT_bChange := 1;
      OUT_rDiff   := rInput - rOld ;
      rOldLimitIn := rLimitIn ;
      rOld := rInput ;
		ELSE
			OUT_bChange := 0;
		END_IF
	ELSE
		OUT_bChange :=0;
	END_IF

  INOUT_rLimitIn := rLimitIn ;

END_FUNCTION_BLOCK
```

#### H_FB_RelativeChangeLimitReal1.st - Detects A Change Of A Real Number For One Scan
```iecst
(********************************************************************
 * COPYRIGHT --
 ********************************************************************
 * Library: HGWeber
 * File: H_FB_RelativeChangeLimitReal.st
 * Author: dominique
 * Created: October 10, 2011
 ********************************************************************
 * Implementation of library HGWeber
 ********************************************************************)

(*Detects A Change Of A Real Number For One Scan and limit the Change*)
FUNCTION_BLOCK H_FB_RelativeChangeLimitReal1

  rMax := IN_rRepeat * IN_rMax ;
  rMin := IN_rRepeat * IN_rMin ;

	OUT_bOK := IN_bEnable;
	IF (IN_bEnable) THEN
    rDiff := IN_rLimitIn - rOldLimitIn ;
    OUT_rLimitIn := IN_rLimitIn ;
    // Limit relative change
    IF rDiff > rMax THEN
      OUT_rLimitIn := rOldLimitIn + rMax ;
    END_IF
    IF rDiff < rMin THEN
      OUT_rLimitIn := rOldLimitIn + rMin ;
    END_IF
    rInput := OUT_rLimitIn + IN_rInput ;
		IF (rInput <> rOld) THEN
			OUT_bChange := 1;
      OUT_rDiff   := rInput - rOld ;
      rOldLimitIn := OUT_rLimitIn ;
      rOld := rInput ;
      iCount := iCount + 1 ;
      IF iCount < 0 THEN
        iCount := 0 ;
      END_IF
		ELSE
			OUT_bChange := 0;
		END_IF
  ELSE;
    OUT_rLimitIn := IN_rLimitIn ;
    rOldLimitIn  := OUT_rLimitIn ;
    rOld         := OUT_rLimitIn + IN_rInput ;
		OUT_bChange  := 0 ;
	END_IF;

END_FUNCTION_BLOCK
```

### Program Logical/SupervisoryControl_Section/Setup (IEC) - Setup Mode Control

#### Setup.var
```iecst
(********************************************************************
 * COPYRIGHT -- Microsoft
 ********************************************************************
 * Program: Setup
 * File: Setup.var
 * Author: pkiel
 * Created: July 20, 2011
 ********************************************************************
 * Local variables of program Setup
 ********************************************************************)
VAR RETAIN
	HGW_2StatePB_0 : HGW_2StatePB;
END_VAR
VAR
	SetupMode_PB : BOOL;
	SetupModeColor_Ind : UINT;
	SetupModeText_Ind : UINT;
	SpeedLimit : INT;

END_VAR
```

#### SetupCyclic.st
```iecst
(********************************************************************
 * COPYRIGHT -- Microsoft
 ********************************************************************
 * Program: Setup
 * File: SetupCyclic.st
 * Author: pkiel
 * Created: July 20, 2011
 ********************************************************************
 * Implementation of program Setup
 ********************************************************************)

PROGRAM _CYCLIC

(* Setup Mode Off/On From HMI *)
	HGW_2StatePB_0.PB := EDGEPOS(SetupMode_PB AND gSetupPermissive);
	SetupModeText_Ind := HGW_2StatePB_0.Text_Ind;
	SetupModeColor_Ind := HGW_2StatePB_0.Color_Ind;
	gSetupMode_On := HGW_2StatePB_0.State1;
	HGW_2StatePB_0();

(* Setup Mode Permissive...Line Speed Must Be <= 10mpm (32.808 fpm) *)
	IF (gActualMachineSpeed_FPM<=32.808) THEN
		gSetupPermissive := 1;
	ELSE
		gSetupPermissive := 0;
	END_IF

(* Setup Mode Guard Bypass Control *)
	IF (gSetupMode_On) THEN
		gQ_CR_GuardBypass := 1;
	ELSE
		gQ_CR_GuardBypass := 0;
	END_IF

// General constants assignment
  // ----------------------------------------
  g_rSizeLPerf_mm         := 400.0 ; // Perimeter of the large Perf, in mm
  g_rSizeSPerf_mm         := 270.0 ; // Perimeter of the small Perf, in mm
  g_rSizeEntryPullRol_mm  := 400.0 ; // Perimeter of the entry pull roll, in mm
  g_rSizeExitPullRol_mm   := 320.0;  // Perimeter of the exit pull roll, in mm
  g_rSizeDrum_mm          := 1680.0; // Perimeter of the Drum, in mm
  g_rZGearRepFP_M         := 40.0 ;  // Tooth number of the gear on the Flexo Press in case Metric
  g_rZGearRepFP_8DP       := 40.0 ;  // Tooth number of the gear on the Flexo Press in case 8DP
  g_rZGearRepFP_10DP      := 50.0 ;  // Tooth number of the gear on the Flexo Press in case 10DP
  g_rZGearRepFP_1_4P      := 65.0 ;  // Tooth number OF the gear on the Flexo Press in CASE 1/4"
  g_rZGearCMPerf_M        := 50.0 ;  // Tooth number of the gear on the shaft which drive the Cold Micro Perf Tool in case Metric
  g_rZGearCMPerf_8DP      := 50.0 ;  // Tooth number of the gear on the shaft which drive the Cold Micro Perf Tool in case 8DP
  g_rZGearCMPerf_10DP     := 63.0 ;  // Tooth number of the gear on the shaft which drive the Cold Micro Perf Tool in case 10DP
  g_rZGearCMPerf_1_4P     := 81.0 ;  // Tooth number of the gear on the shaft which drive the Cold Micro Perf Tool in case 1/4"

  // General parameter init
  gr_rMachMaxSpeed_BPM := 1000.0 ;

  gr_rPosHoldBag := gr_rPosHoldBag ;
  gr_rPosTearBag := gr_rPosTearBag ;
  gr_rPosGripBag := gr_rPosGripBag ;

  gr_rPosEnvBHoldBag   := gr_rPosEnvBHoldBag ;
  gr_rPosTearEBTearBag := gr_rPosTearEBTearBag ;

  // ----------------------------------------
  // Cycles
  // Manual timing setting
  g_rCycManTimSetOverrideAcc := 0.5 ;

END_PROGRAM
```

### Program Logical/SupervisoryControl_Section/ManMode (IEC) - Manual Mode Control

#### ManMode.var
```iecst
(********************************************************************
 * COPYRIGHT -- Microsoft
 ********************************************************************
 * Program: ManMode
 * File: ManMode.var
 * Author: pkiel
 * Created: July 22, 2011
 ********************************************************************
 * Local variables of program ManMode
 ********************************************************************)
VAR RETAIN
	HGW_2StatePB_0 : HGW_2StatePB;
END_VAR
VAR
	ManualDataLock : UINT;
	ManualMode_PB : BOOL;
	ManualModeColor_Ind : UINT;
	ManualModeText_Ind : UINT;
  uiPhasSetLock : UINT;
  uiPhasTearingSetLock : UINT;
END_VAR
```

#### ManModeCyclic.st
```iecst
(********************************************************************
 * COPYRIGHT -- Microsoft
 ********************************************************************
 * Program: ManMode
 * File: ManModeCyclic.st
 * Author: pkiel
 * Created: July 22, 2011
 ********************************************************************
 * Implementation of program ManMode
 ********************************************************************)

PROGRAM _CYCLIC

(* Manual Mode Off/On From HMI *)
	HGW_2StatePB_0.PB := EDGEPOS(ManualMode_PB);
	ManualModeText_Ind := HGW_2StatePB_0.Text_Ind;
	ManualModeColor_Ind := HGW_2StatePB_0.Color_Ind;
	gManualMode_On := HGW_2StatePB_0.State1;
	HGW_2StatePB_0();

(* Manaul Mode Data Lock *)
	IF (gManualMode_On) THEN
		ManualDataLock := 0;
	ELSE
		ManualDataLock := 2;
  END_IF

  // Screen axis phase setting lock
  IF g_bMachineRun       AND
     gManualMode_On      AND
     g_bSynchroAxisOK    AND
     g_bIndPhasDrumInact AND
     1                   THEN
    uiPhasSetLock := 0 ; // Free
  ELSE
    uiPhasSetLock := 2;  // Lock
  END_IF
  uiPhasTearingSetLock := 2 ; // When machine is running not possible to move Tearing axis alone always Holding+Tearing
END_PROGRAM
```

### Program Logical/SupervisoryControl_Section/Speed (IEC) - Main Machine Speed Limit

#### Speed.var
```iecst
(********************************************************************
 * COPYRIGHT -- Microsoft
 ********************************************************************
 * Program: SpeedLimit
 * File: SpeedLimit.var
 * Author: pkiel
 * Created: July 21, 2011
 ********************************************************************
 * Local variables of program SpeedLimit
 ********************************************************************)
VAR
	Ar_iMaxSpeedLargePerf : ARRAY[75..850] OF INT; (*Tab Max Speed Large Perf, in bag/min*)
	Ar_iMaxSpeedSmallPerf : ARRAY[75..850] OF INT; (*Tab Max Speed Small Perf, in bag/min*)
	Ar_iMaxSpeedApPoPerf_520 : ARRAY[75..850] OF INT; (*Tab Max Speed Envelope Bag Perf, in bag/min*)
END_VAR
VAR RETAIN
	ArrayIndex : INT;
END_VAR
VAR
	Index1 : INT;
	PerfCylSelect_Old : BOOL;
	Remainder : REAL;
	RepeatMetric : REAL;
	SpeedLimit : INT;
	rConvAccDec : REAL;
	rLinSpeedSP_JogDec : REAL;
	bIndSynchro_OK : BOOL;
	bLimSpeedSynchro : BOOL;
	uiiMemoNumRev : UDINT;
	uiiDiffNumRev : UDINT;
	bMemoSynchro_OK : BOOL;
	rBundSpeedLimit : REAL;
	rFPSpeedLimit : REAL;
	rBagSize1to2Perf_mm : REAL;
END_VAR
```

### Program Logical/SupervisoryControl_Section/Guard_Mon (IEC) - Guard Monitor Code

#### Guard_MonCyclic.ld
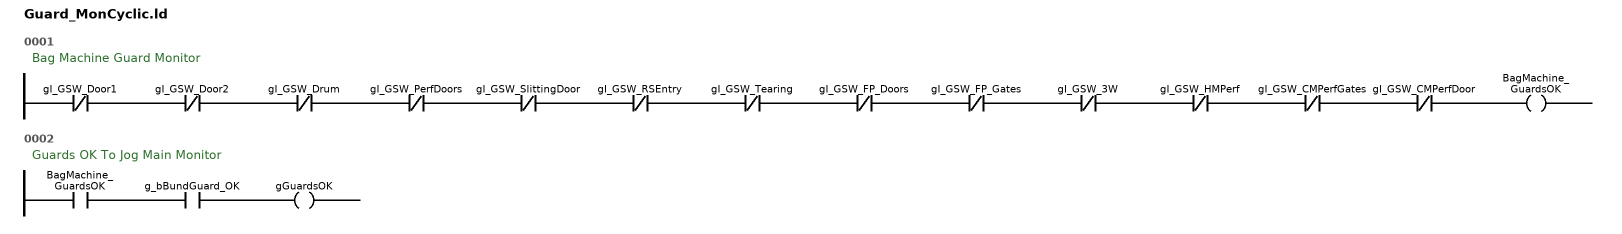
Ladder, written as Structured Text:
```iecst
(********************************************************************
 * COPYRIGHT --
 ********************************************************************
 * Program: Guard_Mon
 * File: Guard_MonCyclic.ld
 * Author: pkiel
 * Created: October 13, 2009
 ********************************************************************
 * Implementation of program Guard_Mon
 ********************************************************************)

PROGRAM _CYCLIC
(* Network 1: Bag Machine Guard Monitor *)
BagMachine_GuardsOK := NOT gI_GSW_Door1 AND NOT gI_GSW_Door2 AND NOT gI_GSW_Drum AND NOT gI_GSW_PerfDoors AND NOT gI_GSW_SlittingDoor AND NOT gI_GSW_RSEntry AND NOT gI_GSW_Tearing AND NOT gI_GSW_FP_Doors AND NOT gI_GSW_FP_Gates AND NOT gI_GSW_3W AND NOT gI_GSW_HMPerf AND NOT gI_GSW_CMPerfGates AND NOT gI_GSW_CMPerfDoor;

(* Network 2: Guards OK To Jog Main Monitor *)
gGuardsOK := BagMachine_GuardsOK AND g_bBundGuard_OK;
END_PROGRAM
```

### Program Logical/SupervisoryControl_Section/Stop_Mon (IEC) - Stop Monitor Code

#### Stop_MonCyclic.ld
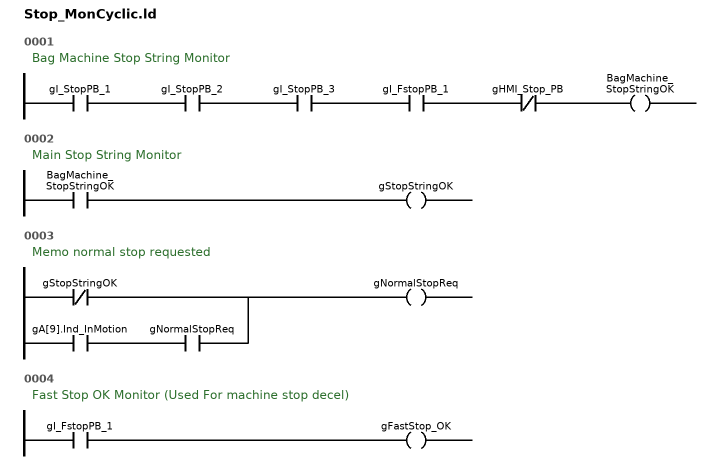
Ladder, written as Structured Text:
```iecst
(********************************************************************
 * COPYRIGHT --
 ********************************************************************
 * Program: Stop_Mon
 * File: Stop_MonCyclic.ld
 * Author: pkiel
 * Created: October 13, 2009
 ********************************************************************
 * Implementation of program Stop_Mon
 ********************************************************************)

PROGRAM _CYCLIC
(* Network 1: Bag Machine Stop String Monitor *)
BagMachine_StopStringOK := gI_StopPB_1 AND gI_StopPB_2 AND gI_StopPB_3 AND gI_FstopPB_1 AND NOT gHMI_Stop_PB;

(* Network 2: Main Stop String Monitor *)
gStopStringOK := BagMachine_StopStringOK;

(* Network 3: Memo normal stop requested *)
gNormalStopReq := NOT gStopStringOK OR (gA[9].Ind_InMotion AND gNormalStopReq);

(* Network 4: Fast Stop OK Monitor (Used For machine stop decel) *)
gFastStop_OK := gI_FstopPB_1;
END_PROGRAM
```

- Program Logical/SupervisoryControl_Section/Servo_Mon (IEC) - Servo Monitor Code (no source held here)

### Program Logical/SupervisoryControl_Section/Alarm_Section/Alarms1 (IEC)

#### Alarms1Init.st - Initialization code
```iecst
(********************************************************************
 * COPYRIGHT -- .
 ********************************************************************
 * Program: Alarms1
 * File: NewProgramInit.st
 * Author: dominique
 * Created: December 09, 2011
 ********************************************************************
 * Implementation of program Alarms1
 ********************************************************************)

PROGRAM _INIT

  bTest := 0 ;
  Alarm1 := Alarm1 ; // D.M. RS26_Pyrollpack_14661 added just to be able to see all items at once in Monitor

END_PROGRAM
```

#### Alarms1.typ - Local data types
```iecst
(********************************************************************
 * COPYRIGHT --
 ********************************************************************
 * Program: Alarms1
 * File: Alarms1.typ
 * Author: pkiel
 * Created: September 22, 2009
 ********************************************************************
 * Local data types of program Alarms1
 ********************************************************************)

TYPE
  stIO_Alarm : STRUCT
      bStat   : BOOL := FALSE ;
      strType : STRING[15] := '' ;
    END_STRUCT;
END_TYPE
```

#### Alarms1.var - Local variables
```iecst
(********************************************************************
 * COPYRIGHT --
 ********************************************************************
 * Program: Alarms1
 * File: Alarms1.var
 * Author: pkiel
 * Created: September 22, 2009
 ********************************************************************
 * Local variables of program Alarms1
 ********************************************************************)
VAR CONSTANT
  C_iMaxAlmIO_E1      : INT := 20 ; (*Max number of modules on the remote IO device*)
  C_iNumBefFirstIO_E1 : INT := 2 ;  (*Number of modules before the first IO module = network + alim modules*)
  C_iNumDI_E1 : INT := 3 ;  (*Number of Digital Input modules*)
  C_iNumAI_E1 : INT := 1 ;  (*Number of Anologe Input modules*)
  C_iNumDO_E1 : INT := 2 ;  (*Number of Digital Output modules*)
  C_iNumAO_E1 : INT := 1 ;  (*Number of Anologe Output modules*)

  C_iMaxAlmIO_L3      : INT := 20 ;
  C_iNumBefFirstIO_L3 : INT := 1 ;
  C_iNumDI_L3 : INT := 4 ;
  C_iNumAI_L3 : INT := 0 ;
  C_iNumDO_L3 : INT := 1 ;
  C_iNumAO_L3 : INT := 1 ;
  C_iX2XExt_L3 : INT := 0 ;

  C_iMaxAlmIO_L9      : INT := 20 ;
  C_iNumBefFirstIO_L9 : INT := 1 ;
  C_iNumDI_L9 : INT := 5 ;
  C_iNumAI_L9 : INT := 1 ;
  C_iNumDO_L9 : INT := 4 ;
  C_iNumAO_L9 : INT := 0 ;
  C_iX2XExt_L9 : INT := 0 ;

  C_iMaxAlmIO_L15      : INT := 20 ;
  C_iNumBefFirstIO_L15 : INT := 1 ;
  C_iNumDI_L15 : INT := 5 ;
  C_iNumAI_L15 : INT := 0 ;
  C_iNumDO_L15 : INT := 1 ;
  C_iNumAO_L15 : INT := 0 ;
  C_iX2XExt_L15 : INT := 0 ;
END_VAR
VAR
  Alarm1 : ARRAY[0..200] OF BOOL := [200(FALSE)];
  BagMachineBitmap1_Ind : UINT;
  bAlarmIO_E1 : ARRAY[0..C_iMaxAlmIO_E1] OF BOOL := [C_iMaxAlmIO_E1(FALSE)];
  bAlarmGenIO_E1 : BOOL ;
  bAlarmIO_L3 : ARRAY[0..C_iMaxAlmIO_L3] OF BOOL := [C_iMaxAlmIO_L3(FALSE)];
  bAlarmGenIO_L3 : BOOL ;
  bAlarmIO_L9 : ARRAY[0..C_iMaxAlmIO_L9] OF BOOL := [C_iMaxAlmIO_L9(FALSE)];
  bAlarmGenIO_L9 : BOOL ;
  bAlarmIO_L15 : ARRAY[0..C_iMaxAlmIO_L15] OF BOOL := [C_iMaxAlmIO_L15(FALSE)];
  bAlarmGenIO_L15 : BOOL ;
  iIndex : INT := 0 ;
  bActOut : BOOL ;
  bBagMachineBitmap1_Ind : UINT;
  BagMachineVisibility1_Ind : UINT;
  EstopString1 : BOOL;
  EstopString2 : BOOL;
  EstopString3 : BOOL;
  GuardAlarmEnable : BOOL;
  HGW_2StateIND1_0 : HGW_2StateIND1;
  IO_String1 : BOOL;
  IO_String2 : BOOL;
  IO_String3 : BOOL;
  IO_String4 : BOOL;
  IO_String5 : BOOL;
  IO_String6 : BOOL;

  stModuleOK_IO_E1_Slot  : ARRAY[0..C_iMaxAlmIO_E1] OF stIO_Alarm ;
  stModuleOK_IO_L3_Slot  : ARRAY[0..C_iMaxAlmIO_L3] OF stIO_Alarm ;
  stModuleOK_IO_L9_Slot  : ARRAY[0..C_iMaxAlmIO_L9] OF stIO_Alarm ;
  stModuleOK_IO_L15_Slot : ARRAY[0..C_iMaxAlmIO_L9] OF stIO_Alarm ;
  MotorString1  : BOOL;
  MotorString2  : BOOL;
  MotorString3  : BOOL;
  MotorString4  : BOOL;
  MotorString5  : BOOL;
  MotorString6  : BOOL;
  MotorString7  : BOOL;
  MotorString8  : BOOL;
  bGuardString1 : BOOL;
  bGuardString2 : BOOL;
  TON_1 : TON;
  TON_2 : TON;
  TON_3 : TON;
  TON_4 : TON;
  TON_5 : TON;
  TON_6 : TON;
  TON_7 : TON;
  TON_8 : TON;
  TON_12 : TON;
  TON_13 : TON;
  TON_15 : TON;
  TON_30 : TON;
  TON_31 : TON;
  TON_32 : TON;
  GuardAlarmEnable1 : BOOL;

  iVisiblES_BP1 : INT ;
  iVisiblES_BP2 : INT ;
  iVisiblES_BP3 : INT ;
  iVisiblES_BP4 : INT ;
  iVisiblES_BP5 : INT ;
  iVisiblES_BP6 : INT ;
  iVisiblES_BP7 : INT ;
  iVisiblES_BP8 : INT ;
  iVisiblES_BP9 : INT ;
  iVisiblES_BP10 : INT ;

  iVisiblSG1 : INT ;
  iVisiblSG2 : INT ;
  iVisiblSG3 : INT ;
  iVisiblSG4 : INT ;
  iVisiblSG5 : INT ;
  iVisiblSG6 : INT ;

  H_FB_Flash_0 : H_FB_Flash ;

  bTest : BOOL := 0 ;
END_VAR
```

### Program Logical/SupervisoryControl_Section/Alarm_Section/EStopReset (IEC)

#### EStopReset.var - Local variables
```iecst
(********************************************************************
 * COPYRIGHT --
 ********************************************************************
 * Program: EStopReset
 * File: EStopReset.var
 * Author: pkiel
 * Created: October 12, 2009
 ********************************************************************
 * Local variables of program EStopReset
 ********************************************************************)
VAR
	ESR_ResetTimer : TON;
	ESR_Reset : BOOL;
END_VAR
```

### Program Logical/SupervisoryControl_Section/Alarm_Section/MainAlarms

#### MainAlarms.var
```iecst
(********************************************************************
 * COPYRIGHT --
 ********************************************************************
 * Program: MainAlarms
 * File: MainAlarms.var
 * Author: pkiel
 * Created: October 13, 2009
 ********************************************************************
 * Local variables of program MainAlarms
 ********************************************************************)
VAR
	AlarmColor_Ind : UINT;
	AlarmScreenActive : BOOL;
	AlarmVisibility_Ind : UINT;
	EStopAlarmColor_Ind : UINT;
	GuardAlarmColor_Ind : UINT;
	HGW_2StateIND_0 : HGW_2StateIND;
	HGW_2StateIND_1 : HGW_2StateIND;
	HGW_2StateIND_2 : HGW_2StateIND;
	HGW_2StateIND_3 : HGW_2StateIND;
  HGW_2StateIND_4 : HGW_2StateIND;
  HGW_2StateIND_5 : HGW_2StateIND;
  HGW_2StateIND_6 : HGW_2StateIND;
	HGW_2StateIND1_0 : HGW_2StateIND1;
	IOAlarmColor_Ind : UINT;
	JamAlarmColor_Ind : UINT;
	LastScreen : UINT;
	LastScreenOK : BOOL;
	MotorAlarmColor_Ind : UINT;
END_VAR
```

#### MainAlarmsCyclic.ld
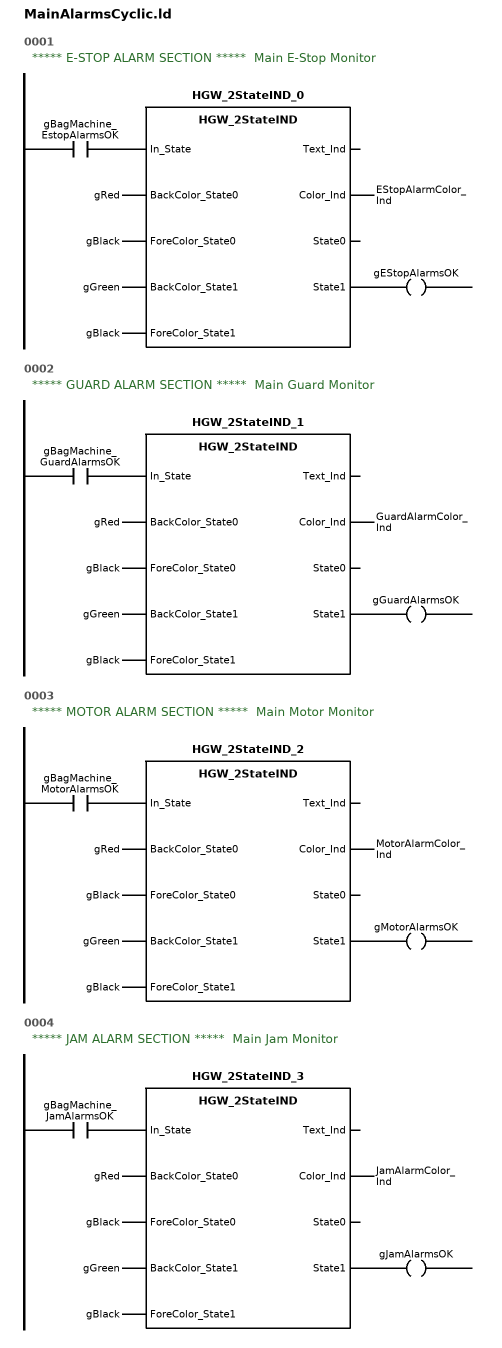
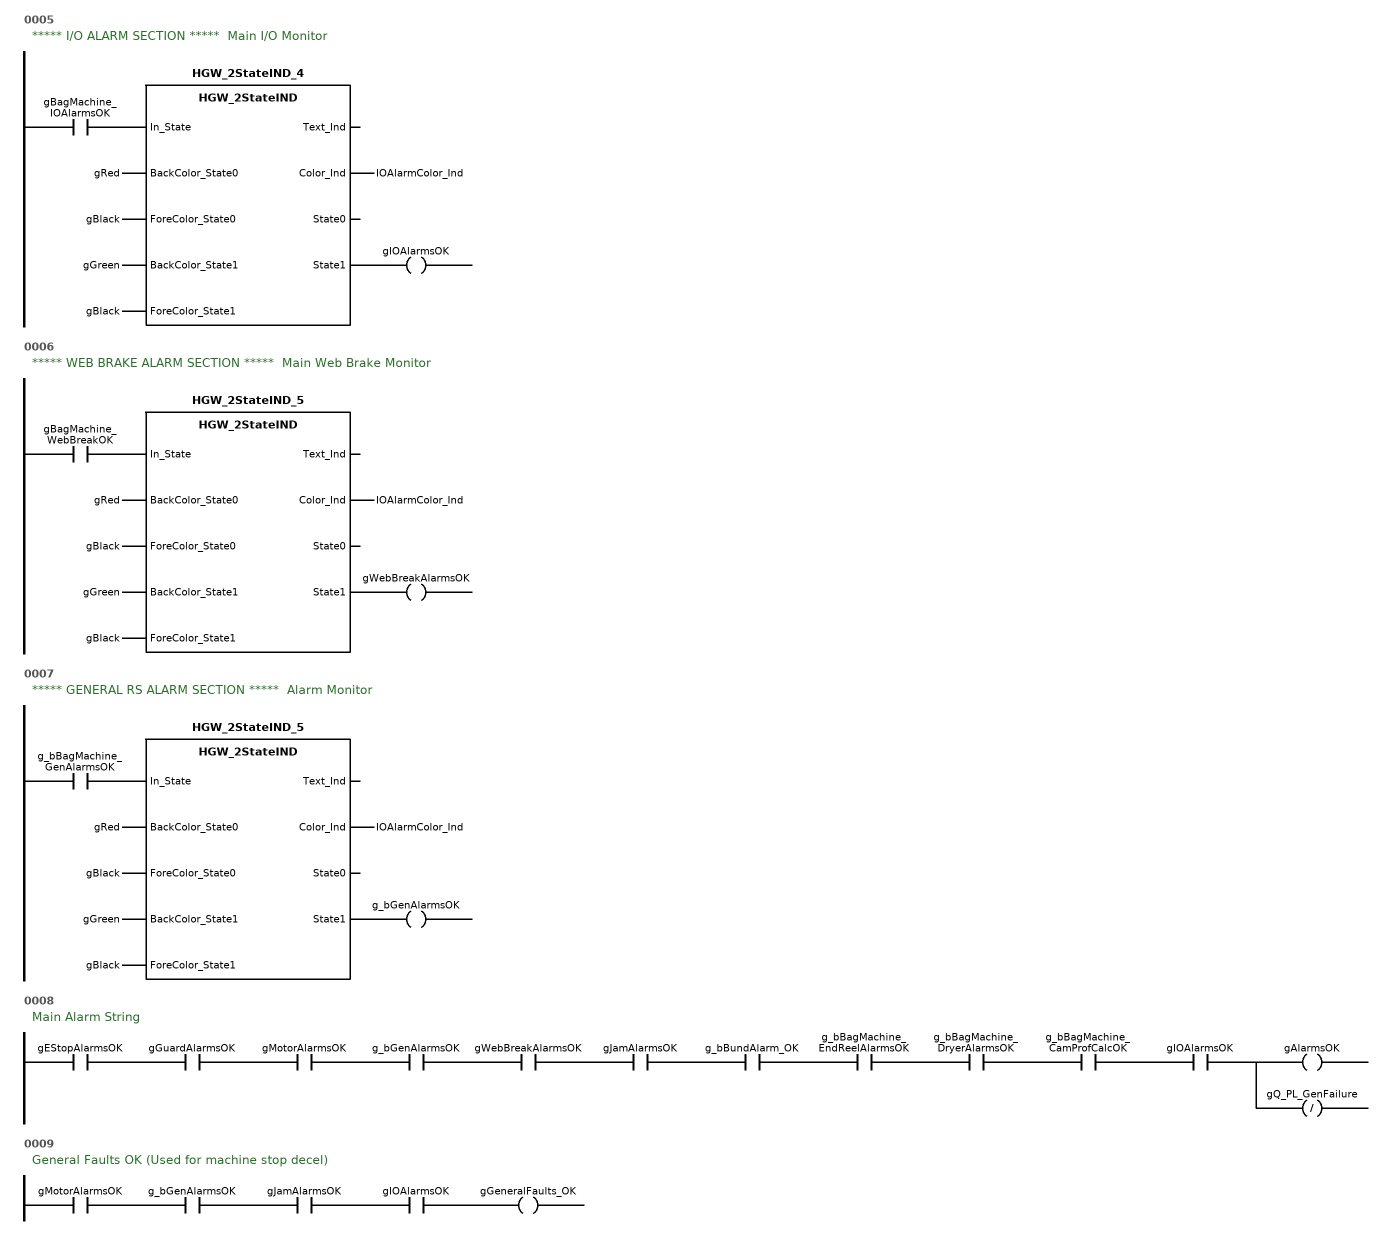
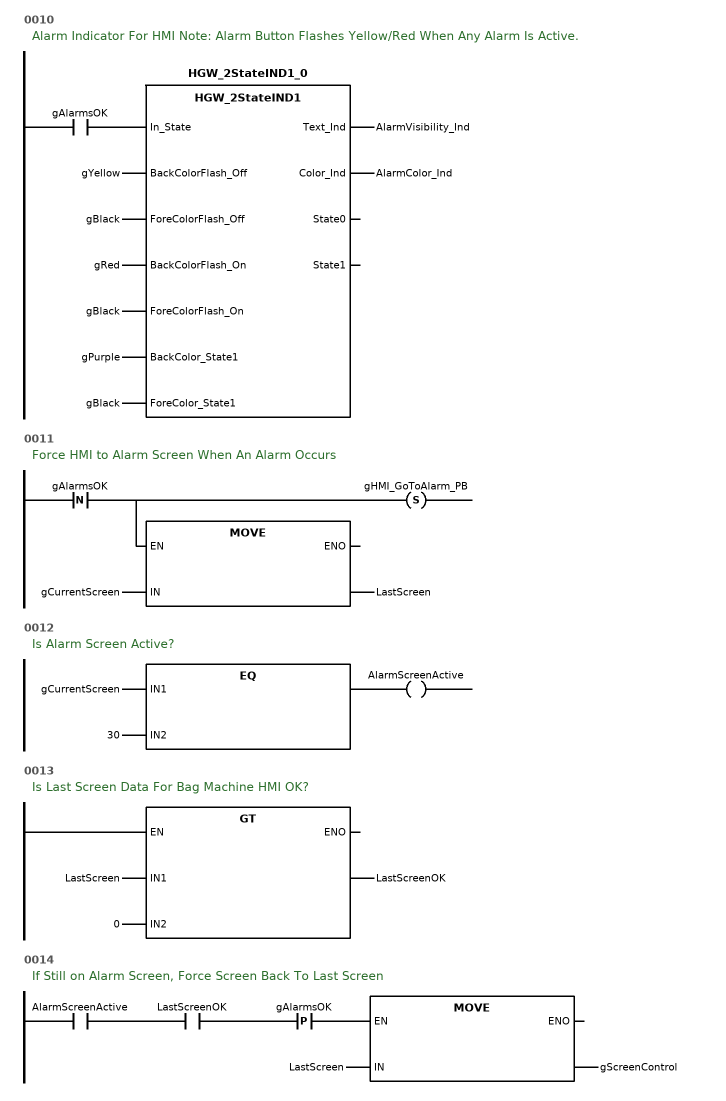
Ladder, written as Structured Text:
```iecst
(********************************************************************
 * COPYRIGHT --
 ********************************************************************
 * Program: MainAlarms
 * File: MainAlarmsCyclic.ld
 * Author: pkiel
 * Created: October 13, 2009
 ********************************************************************
 * Implementation of program MainAlarms
 ********************************************************************)

PROGRAM _CYCLIC
VAR
    _p1 : BOOL;
    _e2 : F_TRIG;
    _e3 : R_TRIG;
END_VAR
(* Network 1: ***** E-STOP ALARM SECTION *****  Main E-Stop Monitor *)
HGW_2StateIND_0(In_State := gBagMachine_EstopAlarmsOK, BackColor_State0 := gRed, ForeColor_State0 := gBlack, BackColor_State1 := gGreen, ForeColor_State1 := gBlack);
EStopAlarmColor_Ind := HGW_2StateIND_0.Color_Ind;
gEStopAlarmsOK := HGW_2StateIND_0.State1;

(* Network 2: ***** GUARD ALARM SECTION *****  Main Guard Monitor *)
HGW_2StateIND_1(In_State := gBagMachine_GuardAlarmsOK, BackColor_State0 := gRed, ForeColor_State0 := gBlack, BackColor_State1 := gGreen, ForeColor_State1 := gBlack);
GuardAlarmColor_Ind := HGW_2StateIND_1.Color_Ind;
gGuardAlarmsOK := HGW_2StateIND_1.State1;

(* Network 3: ***** MOTOR ALARM SECTION *****  Main Motor Monitor *)
HGW_2StateIND_2(In_State := gBagMachine_MotorAlarmsOK, BackColor_State0 := gRed, ForeColor_State0 := gBlack, BackColor_State1 := gGreen, ForeColor_State1 := gBlack);
MotorAlarmColor_Ind := HGW_2StateIND_2.Color_Ind;
gMotorAlarmsOK := HGW_2StateIND_2.State1;

(* Network 4: ***** JAM ALARM SECTION *****  Main Jam Monitor *)
HGW_2StateIND_3(In_State := gBagMachine_JamAlarmsOK, BackColor_State0 := gRed, ForeColor_State0 := gBlack, BackColor_State1 := gGreen, ForeColor_State1 := gBlack);
JamAlarmColor_Ind := HGW_2StateIND_3.Color_Ind;
gJamAlarmsOK := HGW_2StateIND_3.State1;

(* Network 5: ***** I/O ALARM SECTION *****  Main I/O Monitor *)
HGW_2StateIND_4(In_State := gBagMachine_IOAlarmsOK, BackColor_State0 := gRed, ForeColor_State0 := gBlack, BackColor_State1 := gGreen, ForeColor_State1 := gBlack);
IOAlarmColor_Ind := HGW_2StateIND_4.Color_Ind;
gIOAlarmsOK := HGW_2StateIND_4.State1;

(* Network 6: ***** WEB BRAKE ALARM SECTION *****  Main Web Brake Monitor *)
HGW_2StateIND_5(In_State := gBagMachine_WebBreakOK, BackColor_State0 := gRed, ForeColor_State0 := gBlack, BackColor_State1 := gGreen, ForeColor_State1 := gBlack);
IOAlarmColor_Ind := HGW_2StateIND_5.Color_Ind;
gWebBreakAlarmsOK := HGW_2StateIND_5.State1;

(* Network 7: ***** GENERAL RS ALARM SECTION *****  Alarm Monitor *)
HGW_2StateIND_5(In_State := g_bBagMachine_GenAlarmsOK, BackColor_State0 := gRed, ForeColor_State0 := gBlack, BackColor_State1 := gGreen, ForeColor_State1 := gBlack);
IOAlarmColor_Ind := HGW_2StateIND_5.Color_Ind;
g_bGenAlarmsOK := HGW_2StateIND_5.State1;

(* Network 8: Main Alarm String *)
_p1 := gEStopAlarmsOK AND gGuardAlarmsOK AND gMotorAlarmsOK AND g_bGenAlarmsOK AND gWebBreakAlarmsOK AND gJamAlarmsOK AND g_bBundAlarm_OK AND g_bBagMachine_EndReelAlarmsOK AND g_bBagMachine_DryerAlarmsOK AND g_bBagMachine_CamProfCalcOK AND gIOAlarmsOK;
gAlarmsOK := _p1;
gQ_PL_GenFailure := NOT _p1;

(* Network 9: General Faults OK (Used for machine stop decel) *)
gGeneralFaults_OK := gMotorAlarmsOK AND g_bGenAlarmsOK AND gJamAlarmsOK AND gIOAlarmsOK;

(* Network 10: Alarm Indicator For HMI Note: Alarm Button Flashes Yellow/Red When Any Alarm Is Active. *)
HGW_2StateIND1_0(In_State := gAlarmsOK, BackColorFlash_Off := gYellow, ForeColorFlash_Off := gBlack, BackColorFlash_On := gRed, ForeColorFlash_On := gBlack, BackColor_State1 := gPurple, ForeColor_State1 := gBlack);
AlarmVisibility_Ind := HGW_2StateIND1_0.Text_Ind;
AlarmColor_Ind := HGW_2StateIND1_0.Color_Ind;

(* Network 11: Force HMI to Alarm Screen When An Alarm Occurs *)
_e2(CLK := gAlarmsOK);
IF _e2.Q THEN
    gHMI_GoToAlarm_PB := TRUE;
    LastScreen := gCurrentScreen;
END_IF;

(* Network 12: Is Alarm Screen Active? *)
AlarmScreenActive := gCurrentScreen = 30;

(* Network 13: Is Last Screen Data For Bag Machine HMI OK? *)
LastScreenOK := LastScreen > 0;

(* Network 14: If Still on Alarm Screen, Force Screen Back To Last Screen *)
_e3(CLK := gAlarmsOK);
IF AlarmScreenActive AND LastScreenOK AND _e3.Q THEN gScreenControl := LastScreen; END_IF;
END_PROGRAM
```

### Program Logical/SupervisoryControl_Section/Jog (IEC) - Machine Jog Code

#### Jog.var
```iecst
(********************************************************************
 * COPYRIGHT --
 ********************************************************************
 * Program: Jog
 * File: Jog.var
 * Author: pkiel
 * Created: October 13, 2009
 ********************************************************************
 * Local variables of program Jog
 ********************************************************************)
VAR
	JogPermissives_OK : BOOL;
	HGW_2StepMove_0 : HGW_2StepMove1;
	JogRequest : BOOL;
	AnyJog : BOOL;
	TOF_0 : TOF;
  bMemoMachineJog : BOOL ;
  HGW_2StepMove1_0 : HGW_2StepMove1;
  HGW_2StepMove1_1 : HGW_2StepMove1;
  HGW_2StepMove1_2 : HGW_2StepMove1;
END_VAR
```

### Program Logical/SupervisoryControl_Section/Run (IEC) - Machine Run Code

#### RunCyclic.ld - Cyclic code
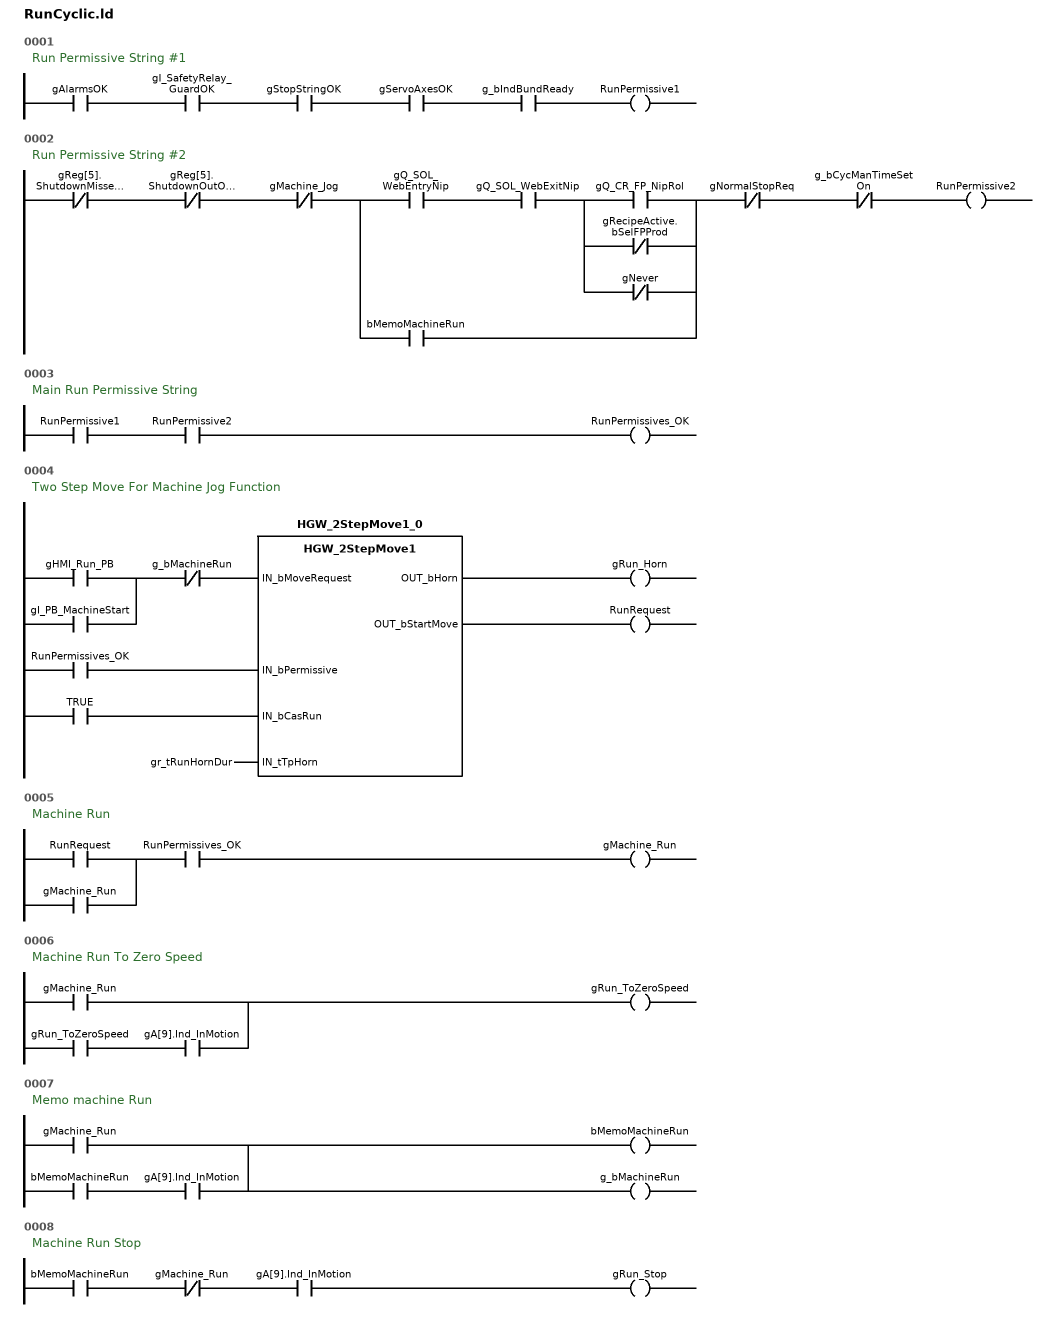
Ladder, written as Structured Text:
```iecst
(********************************************************************
 * COPYRIGHT --
 ********************************************************************
 * Program: Run
 * File: RunCyclic.ld
 * Author: pkiel
 * Created: October 13, 2009
 ********************************************************************
 * Implementation of program Run
 ********************************************************************)

PROGRAM _CYCLIC
VAR
    _p1 : BOOL;
    _p2 : BOOL;
END_VAR
(* Network 1: Run Permissive String #1 *)
RunPermissive1 := gAlarmsOK AND gI_SafetyRelay_GuardOK AND gStopStringOK AND gServoAxesOK AND g_bIndBundReady;

(* Network 2: Run Permissive String #2 *)
_p1 := NOT gReg[5].ShutdownMissedMark AND NOT gReg[5].ShutdownOutOfTolerance AND NOT gMachine_Jog;
RunPermissive2 := _p1 AND ((gQ_SOL_WebEntryNip AND gQ_SOL_WebExitNip AND (gQ_CR_FP_NipRol OR NOT gRecipeActive.bSelFPProd OR NOT gNever)) OR bMemoMachineRun) AND NOT gNormalStopReq AND NOT g_bCycManTimeSetOn;

(* Network 3: Main Run Permissive String *)
RunPermissives_OK := RunPermissive1 AND RunPermissive2;

(* Network 4: Two Step Move For Machine Jog Function *)
HGW_2StepMove1_0(IN_bMoveRequest := (gHMI_Run_PB OR gI_PB_MachineStart) AND NOT g_bMachineRun, IN_bPermissive := RunPermissives_OK, IN_bCasRun := TRUE, IN_tTpHorn := gr_tRunHornDur);
gRun_Horn := HGW_2StepMove1_0.OUT_bHorn;
RunRequest := HGW_2StepMove1_0.OUT_bStartMove;

(* Network 5: Machine Run *)
gMachine_Run := (RunRequest OR gMachine_Run) AND RunPermissives_OK;

(* Network 6: Machine Run To Zero Speed *)
gRun_ToZeroSpeed := gMachine_Run OR (gRun_ToZeroSpeed AND gA[9].Ind_InMotion);

(* Network 7: Memo machine Run *)
_p2 := bMemoMachineRun AND gA[9].Ind_InMotion;
bMemoMachineRun := gMachine_Run OR (bMemoMachineRun AND gA[9].Ind_InMotion);
g_bMachineRun := gMachine_Run OR _p2;

(* Network 8: Machine Run Stop *)
gRun_Stop := bMemoMachineRun AND NOT gMachine_Run AND gA[9].Ind_InMotion;
END_PROGRAM
```

#### Run.var - Local variables
```iecst
(********************************************************************
 * COPYRIGHT --
 ********************************************************************
 * Program: Run
 * File: Run.var
 * Author: pkiel
 * Created: October 13, 2009
 ********************************************************************
 * Local variables of program Run
 ********************************************************************)
VAR
	RunPermissive1 : BOOL;
	RunPermissive2 : BOOL;
	RunPermissives_OK : BOOL;
	RunRequest : BOOL;
	HGW_2StepMove1_0 : HGW_2StepMove1;
  bMemoMachineRun : BOOL;
END_VAR
```

- Program Logical/SupervisoryControl_Section/PowerTimer (IEC) - Startup Power Timer (no source held here)

### Program Logical/SupervisoryControl_Section/HourMeter (IEC) - Tracks Machine Run Time

#### HourMeterCyclic.st
```iecst
(********************************************************************
 * COPYRIGHT --
 ********************************************************************
 * Program: HourMeter
 * File: HourMeterCyclic.st
 * Author: pkiel
 * Created: December 04, 2009
 ********************************************************************
 * Implementation of program HourMeter
 ********************************************************************)

PROGRAM _CYCLIC

(* NOTE: This cyclic program must be run in a 1 second class task to operate properly! *)

	(* Track Machine Run/Jog Time *)
	IF (gMachine_Run OR gMachine_Jog) THEN
		gMachineTime.Seconds := gMachineTime.Seconds+1;
		IF (gMachineTime.Seconds>=60) THEN
			gMachineTime.Minutes := gMachineTime.Minutes + 1;
			gMachineTime.Seconds := 0;
			IF (gMachineTime.Minutes>=60) THEN
				gMachineTime.Hours := gMachineTime.Hours +1;
				gMachineTime.Minutes := 0;
			END_IF
		END_IF
	END_IF

	HourMeterDisplay := DINT_TO_REAL(gMachineTime.Hours)+((INT_TO_REAL(gMachineTime.Minutes))/60.0);

END_PROGRAM
```

- Program Logical/SupervisoryControl_Section/Revision (IEC) - Software Revision Number/Notes (no source held here)

### Program Logical/SupervisoryControl_Section/Warn_Horn (IEC) - A new program

#### Warn_HornCyclic.ld - Cyclic code
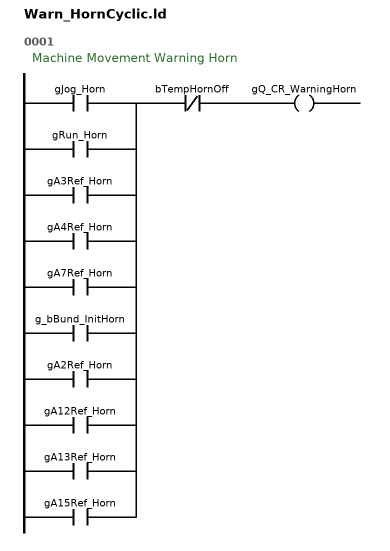
Ladder, written as Structured Text:
```iecst
(********************************************************************
 * COPYRIGHT -- .
 ********************************************************************
 * Program: Warn_Horn
 * File: Warn_HornCyclic.ld
 * Author: dominique
 * Created: August 27, 2011
 ********************************************************************
 * Implementation of program Warn_Horn
 ********************************************************************)

PROGRAM _CYCLIC
(* Network 1: Machine Movement Warning Horn *)
gQ_CR_WarningHorn := (gJog_Horn OR gRun_Horn OR gA3Ref_Horn OR gA4Ref_Horn OR gA7Ref_Horn OR g_bBund_InitHorn OR gA2Ref_Horn OR gA12Ref_Horn OR gA13Ref_Horn OR gA15Ref_Horn) AND NOT bTempHornOff;
END_PROGRAM
```

Listed in the project but not available here: Logical/BagMachine_Section/BagBundler/Control/ControlInit.st, Logical/BagMachine_Section/BagBundler/Control/Control.var, Logical/BagMachine_Section/ColdMicroPerf/Axis8/A8_Basic/A8_BasicCyclic.st, Logical/BagMachine_Section/ColdMicroPerf/Axis8/A8_Basic/A8_Basic.typ, Logical/BagMachine_Section/ColdMicroPerf/CMPerf_Gen/CMPerf_GenInit.st, Logical/BagMachine_Section/ColdMicroPerf/CMPerf_Gen/CMPerf_Gen.var, Logical/BagMachine_Section/Count/CountCyclic.st, Logical/BagMachine_Section/Count/CountInit.st, Logical/BagMachine_Section/Count/Count.typ, Logical/BagMachine_Section/Count/Count.var, Logical/BagMachine_Section/Drum/Axis7/A7_Par, Logical/BagMachine_Section/Drum/Axis7/A7_Basic/A7_BasicInit.st, Logical/BagMachine_Section/Drum/Axis7/A7_Basic/A7_Basic.typ, Logical/BagMachine_Section/EntryPull/Registration/A5_Reg1/A5_Reg1Init.st, Logical/BagMachine_Section/EntryPull/Registration/A5_Reg2/A5_Reg2.var, Logical/BagMachine_Section/EnvBag/Axis12/A12_Control/A12_Control.var, Logical/BagMachine_Section/EnvBag/Axis13/A13_Par, Logical/BagMachine_Section/EnvBag/Axis13/A13_Automat/A13_AutomatCyclic.st, Logical/BagMachine_Section/EnvBag/Axis13/A13_Automat/A13_Automat.var, Logical/BagMachine_Section/EnvBag/Axis13/A13_Ref/A13_Ref.var, Logical/BagMachine_Section/EnvBag/Axis13/A13_Cycle, Logical/BagMachine_Section/EnvBag/EB_Gen/EB_GenCyclic.st, Logical/BagMachine_Section/EnvBag/EB_Gen/EB_GenInit.st, Logical/BagMachine_Section/ExitPull/Axis6/A6_Par, Logical/BagMachine_Section/ExitPull/Axis6/A6_Automat/A6_AutomatCyclic.st, Logical/BagMachine_Section/ExitPull/Axis6/A6_Automat/A6_Automat.typ, Logical/BagMachine_Section/ExitTable/TableCyclic.st, Logical/BagMachine_Section/ExitTable/TableInit.st, Logical/BagMachine_Section/ExitTable/ExitTable.var, Logical/BagMachine_Section/FP/Axis2/A2_Control/A2_ControlCyclic.ld, Logical/BagMachine_Section/FP/Axis2/A2_Control/A2_Control.var, Logical/BagMachine_Section/FP/Axis2/A2_Cycle/A2_CycleCyclic.st, Logical/BagMachine_Section/FP/Axis2/A2_Ref/A2_RefCyclic.ld, Logical/BagMachine_Section/FP/FP_Gen/FP_Gen.typ, Logical/BagMachine_Section/GlobProgCalc/GlobProgCalcInit.st, Logical/BagMachine_Section/Holding/Axis3/A3_Control/A3_Control.var, Logical/BagMachine_Section/HotGlue/HotGlueInit.st, Logical/BagMachine_Section/HotGlue/HotGlue.typ, Logical/BagMachine_Section/HotGlue/HotGlue.var, Logical/BagMachine_Section/HotMicroPerf/Axis15/A15_Automat/A15_AutomatCyclic.st, Logical/BagMachine_Section/HotMicroPerf/Axis15/A15_Automat/A15_Automat.var, Logical/BagMachine_Section/HotMicroPerf/Axis15/A15_Basic/A15_BasicCyclic.st, Logical/BagMachine_Section/HotMicroPerf/Axis15/A15_Basic/A15_Basic.var, Logical/BagMachine_Section/HotMicroPerf/Axis15/A15_MotionCycle/A15_MotionCycleCyclic.st, Logical/BagMachine_Section/MasterAxis/A9_Init/A9_Par, Logical/BagMachine_Section/MasterAxis/A9_Init/A9_Basic/A9_BasicInit.st, Logical/BagMachine_Section/MasterAxis/A9_Init/A9_Control/A9_Control.typ, Logical/BagMachine_Section/MasterAxis/A9_Init/SetSpeedMode/SetSpeedModeCyclic.st, Logical/BagMachine_Section/MasterAxis/A9_Init/SetSpeedMode/SetSpeedModeInit.st, Logical/BagMachine_Section/Perf/Perf_Gen/Perf_Gen.var, Logical/BagMachine_Section/Perf/Perf_Gen/Perf_Gen.typ, Logical/BagMachine_Section/Perf/Axis1/A1_Par, Logical/BagMachine_Section/Perf/Axis1/A1_Control/A1_ControlCyclic.ld, Logical/BagMachine_Section/Perf/Axis1/A1_Control/A1_Control.typ, Logical/BagMachine_Section/Perf/Axis1/A1_Ref/A1_RefCyclic.ld, Logical/BagMachine_Section/Perf/Axis1/A1_Ref/A1_Ref.typ, Logical/BagMachine_Section/Perf/Axis1/A1_CamProfCalc/A1_CamProfCalcCyclic.st, Logical/BagMachine_Section/Perf/Axis1/A1_CamProfCalc/A1_CamProfCalc.var, Logical/BagMachine_Section/Perf/Axis11_VirtualAxis/A11_Basic/A11_BasicCyclic.st, Logical/BagMachine_Section/Perf/Axis11_VirtualAxis/A11_Basic/A11_BasicInit.st, Logical/BagMachine_Section/Perf/Axis11_VirtualAxis/A11_Basic/A11_Basic.typ, Logical/BagMachine_Section/Perf/Axis11_VirtualAxis/A11_Basic/A11_Basic.var, Logical/BagMachine_Section/Tearing/Axis4/A4_Automat/A4_AutomatCyclic.st, Logical/BagMachine_Section/Tearing/Axis4/A4_Automat/A4_Automat.var, Logical/BagMachine_Section/Tearing/Axis4/A4_Cycle/A4_CycleCyclic.st, Logical/BagMachine_Section/Tearing/Axis4/A4_Cycle/A4_CycleInit.st, Logical/BagMachine_Section/Tearing/Axis4/A4_Cycle/A4_Cycle.typ, Logical/BagMachine_Section/Tearing/Axis4/A4_Cycle/A4_Cycle.var, Logical/BagMachine_Section/Unw_3W_Glue/Unw_3W_GlueCyclic.st, Logical/BagMachine_Section/Vacuum/VacuumCyclic.st, Logical/Cycles/GenCycles.var, Logical/HMI/BackUp/BackUpInit.st, Logical/HMI/BackUp/BackUp.typ, Logical/HMI/Cmd_Trace/Cmd_TraceCyclic.st, Logical/HMI/Cmd_Trace/Cmd_Trace.typ, Logical/HMI/Cmd_Trace/Cmd_Trace.var, Logical/HMI/Message_1/Message_1Cyclic.ld, Logical/HMI/Message_1/Message_1.typ, Logical/HMI/Message_1/Message_1.var, Logical/HMI/Message_2/Message_2Cyclic.ld, Logical/HMI/Message_2/Message_2.var, Logical/HMI/Password/PasswordCyclic.st, Logical/HMI/Recipe_1/Recipe_1Cyclic.st, Logical/HMI/Recipe_1/Recipe_1Init.st, Logical/HMI/Recipe_1/Recipe_1.var, Logical/HMI/Recipe_2/Recipe_2Cyclic.st, Logical/HMI/Recipe_2/Recipe_2Init.st, Logical/HMI/Recipe_2/Recipe_2.typ, Logical/HMI/Splash/SplashCyclic.st, Logical/HMI/Splash/Splash.typ, Logical/HMI/Units/Units.typ, Logical/HMI/Units/Units.var, Logical/Information/InformationCyclic.st, Logical/Libraries/HGWeber/HGW_3StatePB.st, Logical/Libraries/HGWeber/HGW_4StatePB.st, Logical/Libraries/HGWeber/HGW_2StateIND.st, Logical/Libraries/HGWeber/HGW_3StateIND.st, Logical/Libraries/HGWeber/HGW_4StateIND.st, Logical/Libraries/HGWeber/HGW_Toggle.ld, Logical/Libraries/HGWeber/HGW_2StepMove.ld, Logical/Libraries/HGWeber/HGW_ScaleReal.st, Logical/Libraries/HGWeber/HGW_KeyRepeat.st, Logical/Libraries/HGWeber/H_FC_Modulus_V0.st, Logical/Libraries/HGWeber/H_FB_2StepMove.st, Logical/Libraries/HGWeber/H_FB_ToggleTB.st, Logical/Libraries/HGWeber/H_FB_WatchSensor.st, Logical/Libraries/HGWeber/H_FC_Modulus.st, Logical/SupervisoryControl_Section/Servo_Mon/Servo_MonCyclic.ld, Logical/SupervisoryControl_Section/Servo_Mon/Servo_Mon.typ, Logical/SupervisoryControl_Section/Servo_Mon/Servo_Mon.var, Logical/SupervisoryControl_Section/Alarm_Section/Alarms1/Alarms1Cyclic.ld, Logical/SupervisoryControl_Section/Alarm_Section/Alarms1/actIO_Ex_FailDetect_E1_L3.st, Logical/SupervisoryControl_Section/Alarm_Section/Alarms1/actIO_Ex_FailDetect_L9.st, Logical/SupervisoryControl_Section/Alarm_Section/Alarms1/actIO_Ex_FailDetect_L15.st, Logical/SupervisoryControl_Section/Alarm_Section/Alarms1/actAnimAlarmVisu.st, Logical/SupervisoryControl_Section/Alarm_Section/EStopReset/EStopResetCyclic.ld, Logical/SupervisoryControl_Section/Alarm_Section/EStopReset/EStopReset.typ, Logical/SupervisoryControl_Section/Run/Run.typ, Logical/SupervisoryControl_Section/PowerTimer/PowerTimerCyclic.ld, Logical/SupervisoryControl_Section/PowerTimer/PowerTimer.var, Logical/SupervisoryControl_Section/Warn_Horn/Warn_HornInit.ld, Logical/SupervisoryControl_Section/Warn_Horn/Warn_Horn.var
